{attribute 'GeneratedUsingTerminal: EM7004-0000-9995'}
{attribute addProperty BoxType "EM7004-0000-9995"}
{attribute addProperty Id "OutputAT %Q*ARRAY[0..15] OF BOOL16"}
{attribute addProperty CRC "1538723034"}
{attribute addProperty Size "16"}
TYPE Digital_A7E1DFAB :
STRUCT
	{attribute addProperty Name "Output"}
	Output AT %Q* : ARRAY[0..15] OF BOOL;
END_STRUCT
END_TYPE
